// TIA Portal V17 export
// export: Created 2024-08-09T12:53:15.2534621Z, ExportSetting WithDefaults, DisplayName Totally Integrated Automation Portal, DisplayVersion V17 Update 7, DisplayName TIA Portal Openness, DisplayVersion V17 Update 7, DisplayName TIA Portal Version Control Interface, DisplayVersion V17, DisplayName STEP 7 Professional, DisplayVersion V17 Update 7, DisplayName STEP 7 Safety, DisplayVersion V17 Update 6, DisplayName WinCC Professional, DisplayVersion V17 Update 7
VAR_GLOBAL   // PLC tag table "Dec_Niveaux_ChargCompo"
END_VAR
VAR_GLOBAL CONSTANT   // user constants
   NIV_CHARGCOMPO_ATT_PREREMP : USInt := 10;
   NIV_CHARGCOMPO_PREREMP : USInt := 15;
   NIV_CHARGCOMPO_ATT_DEM_CIR : USInt := 20;
   NIV_CHARGCOMPO_DEM_CIR : USInt := 30;
   NIV_CHARGCOMPO_CHARG_EC : USInt := 40;
   NIV_CHARGCOMPO_VID_CIR : USInt := 60;
   NIV_CHARGCOMPO_FVID_CIR : USInt := 160;
   NIV_CHARGCOMPO_ATT_FINLOT : USInt := 200;
END_VAR
